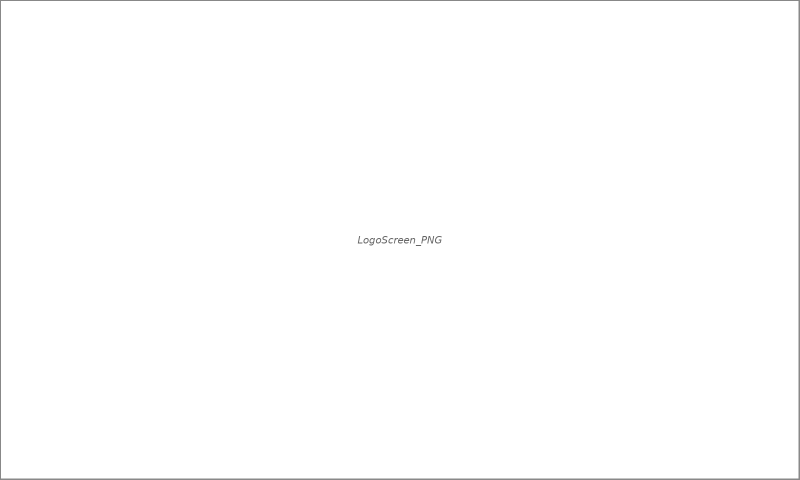
VISUALIZATION Idle_PNG  // 800x480
VAR_IN_OUT
	nUnitsProduced	: UDINT ;
END_VAR
    Frame (0,0 800x480)
        shows LogoScreen_PNG(nUnitsProduced := nUnitsProduced, bCmdManual := GVL_HMI.bCmdManual)
END_VISUALIZATION

(* stored: Version 1.1.0.1, ProductVersion 3.1.4024.9
   Visu Idle_PNG: Id {ceaa85bd-96f6-4a17-821b-25d21a8d47d3} *)
